//****************************************************************************************************
// Code generated by SFC Generator V1.13 on 13/03/19 17:24:34 by  David Paspa from File G:\Business\Synertec\MPI.SMS\automation\code\awlMaster\stencil\seq_hdr.awl
//****************************************************************************************************
//****************************************************************************************************

//================================ SEQ HEADER ================================//
//            Copyright 2018 Rieckermann Engineering Operations               //
//----------------------------------------------------------------------------//
// Title: UO_MX_SIP                                                       //
//                                                                            //
// Description:                                                               //
// Sequence for Mx sterilise in place operation                                                        //
//                                                                            //
// // SFC Revision History:
// Rev By               Date        CC         Note
// 2.0 David Paspa      27-Nov-2018            Reboot for S7-1500
// 0.3 Srinivas Nimmala 19-May-2010            Wong(Changed Cooling-Preempt)
// 0.2 David Paspa      26-Oct-2009            Added synch flags
// 0.1 Gerald Kontriner 09-Sep-2009            SFC structural design                                                       //
//----------------------------------------------------------------------------//
// Sequencer Revision History:                                                //
// Rev By               Date        CC        Note                            //
// 2.0 David Paspa      05-Jan-2018 NA        Reboot for S7-1500.             //
// 1.6 Khairul Basar    19-Nov-2009 NA        Reset #sqSequencer.STEP.Active  //
//                                            when STEP Finished.             //
// 1.5 Khairul Basar    15-Oct-2009 NA        Placeholder inserted:           //
//                                            "udtSQ_UO";          //
// 1.4 Khairul Basar    06-Oct-2009 NA        R #PAUSE;                       //
// 1.3 Khairul Basar    30-Sep-2009 NA        SEQ_HDR change STEP-0 code      //
//                                            deleted.                        //
// 1.2 Khairul Basar    26-Sep-2009 NA        Refer R4.                       //
// 1.1 Khairul Basar    23-Sep-2009 NA        Refer R3.                       //
// 1.0 Khairul Basar    20-Sep-2009 NA        STEP.Finished flag reset by     //
//                                            JUMP_MAN.                       //
// 0.9 Khairul Basar    11-Sep-2009 NA        SQ_TIMER added as VAR, declared //
//                                            in SEQ_FTR.                     //
// 0.8 Khairul Basar    09-Sep-2009 NA        SqSequencer.Err_Fault is reset  //
//                                            on Stop cmd, Step-0 dead code   //
//                                            deleted from ACT & Verify.      //
//                                            STP_FTR Step_withErr flag       //
//                                            STEP_NUM place holder           //
//                                            configured.                     //
// 0.7 Khairul Basar    28-Aug-2009 NA        SQ_FINISHED OUT added again.    //
//                                            Deleted during major mod R3.    //
// 0.6 Khairul Basar    23-Aug-2009 NA        Refer R2.                       //
// 0.5 Khairul Basar    23-Aug-2009 NA        Refer R1.                       //
// 0.4 Khairul Basar    18-Aug-2009 NA        Reset Step done with/out error  //
//                                            bits using FC:RSET.             //
// 0.3 David Paspa      16-Aug-2009 NA        Added placeholders for header   //
//                                            name and version and revision   //
//                                            history.                        //
// 0.2 Khairul Basar    11-Aug-2009 NA        Retired external udt file for   //
//                                            Static type parameters. All     //
//                                            parameters now IN, OUT or       //
//                                            IN_OUT.                         //
// 0.1 Khairul Basar    12-Jun-2009 NA        Initial design.                 //
//----------------------------------------------------------------------------//
// R4:                                                                        //
// 1.If SQ not finished Resume command will start Step timer, and redo the    //
// last action, verify the feedback.                                          //
// 2."STEP.finished" flag is ANDed with "TRN_AND_JUMP" in the snippet file    //
// TRN_HDR.This is to avoid checking of transition logic if STEP is not       //
// finished yet.                                                              //
// 3.MDCH, Load & transfer typo corrected.                                    //
//                                                                            //
// R3:                                                                        //
// 1.SqStepTimer.IN is reset in STEP_FTR instead of resetting it in TRN_HDR.  //
// This is because TRN_HDTR is not included in the Last step and StepTimer    //
// must reset in the last step.                                               //
// 2.Reset all the timers when SQ stops.Reset done in SEQ_HDR.                //
// Also STEP-finished flag reset when SQ is OFF to                            //
// scan last step.                                                            //
//                                                                            //
// R2:                                                                        //
// 1.Any step error will send the Sequencer into Pause state.Code added in    //
// SEQ_HDR.Snippet Place holder for Bool-array 32 is   //
// deleted.                                                                   //
//                                                                            //
// R1:                                                                        //
// 1.sqStepTimer:All Verification Code must satisfy the condition finish step //
// action within STEP_DELAY time(40s).If step actions not finished within the //
// time period the error flag will raise High signal.Else timer will reset.   //
// 2.sqRunTimer Added therefore can be used as retentive & non retentive.     //
// 3.sqSequencer: This is re-structured UDT which is redefined the symbol     //
// names as well as it gives more clearity.                                   //
// 4.fcMODE and fcCMD functions are added to handle the mode & command        //
// independently regardless of other logic.Two separate UDT udtMODE & udt     //
// CMD assigned to Mode & command function respectively.                      //
// 5.MAN_JUMP programed for manual mode jump operation with or without        //
// Transition code satisfied.TRN_AND_JUMP & NO_VERIFC are the parameters      //
// which will define whether verification code & transition code need to be   //
// checked to perform jump operation.                                         //
// 6.Auto to Manual switchover will be bumpless & will not affect step        //
// operation.Manual to auto switchover can be used to resume Step action at   //
// defined.                                                                   //
// Step number entered in STEPNO_JUMP.                                        //
//                                                                            //
// Parameters:                                                                //
// INPUTS                                                                     //
// ======                                                                     //
// SQ_CMD          Sequence command input inherited from object block         //
//                 0: off/idle                                                //
//                 1: start/initiate                                          //
//                 2: pause                                                   //
//                 3: resume                                                  //
//                 4: reserved (not programmed)                               //
//                 5: reserved (not programmed)                               //
//                 6: abort/go to last step                                   //
//                 7: acknowledge error/fault                                 //
// SQ_MODE         Sequencer Auto/Manual input inherited from object block    //
//                 1: manual                                                  //
//                 2: auto                                                    //
//                                                                            //
// INPUT/OUTPUTS                                                              //
// =============                                                              //
// SQ_JUMP_MAN     Allows manual jumping from one step to the next step. The  //
//                 manual jump flag is ORed with the transition process       //
//                 condition and so can be used to bypass the condition if the//
//                 sequence will not progress.                                //
//                 This input can also be used to jump to any step even       //
//                 when no transition -> step linkage exists. This is only    //
//                 possible when the SQ_MODE is in manual and SQ is in the    //
//                 idle step. The step to jump to is specified in             //
//                 SQ_man_jump_to_step (not accesseble by this FB in/out      //
//                 interface but a separate DB memory location).              //
//                                                                            //
// OUTPUTS                                                                    //
// =======                                                                    //
// SQ_STATE        The calculated state of the sequence                       //
//                 0: off/idle                                                //
//                 1: start/initiated                                         //
//                 2: paused                                                  //
//                 3: resumed                                                 //
//                 4: reserved (wrong Mode)                                   //
//                 5: reserved (Wrong commad)                                 //
//                 6: aborted/go to last step                                 //
//                 7: acknowledged error/fault                                //
// CURSTEP         Current step being proccessed.                             //
// S_ACTIVE        If current step is active                                  //
// NXT_STEP        Next step to jump to if transition condition is true       //
// ERR_FAULT       True if any error/ or fault present                        //
// PAUSED          True if step is paused                                     //
// OFF_IDLE        Sequence is not running but ready for next SQ (in step=0)  //
//----------------------------------------------------------------------------//
// Define variables:                                                          //
//----------------------------------------------------------------------------//
FUNCTION_BLOCK "fbUO_MX_SIP"
TITLE = UO : MX_SIP
{ S7_Optimized_Access := 'TRUE' }
NAME : MUSIP
AUTHOR : REO
VERSION : 2.0

VAR_IN_OUT
    _emv_inlet_state :INT ;	//Vessel inlet sprayballs state
    _vessel_mx :INT ;	//Manufacturing vessel selection M1 or M2
    _emc_gas_pi_vessel_pv :REAL ;	//Vessel pressure
    _emx_drain_state :INT ;	//Device state of emx_drain
    _ema_vessel_state :INT ;	//Device State of ema_vessel
    _emx_mmfl_state :INT ;	//Device state of emx_mmfl
    _emv_vessel_ti_vessel_pv :REAL ;	//TIn105 Vessel Temperature
    _emg_filter_ti_drain_pv :REAL ;	//TIn103 Vent Filter Top Outlet Temperature
    _emt_hex_ti_hex_pv :REAL ;	//TIn109 Heat Exchanger Outlet Temperature
    _emx_drain_ti_drain_pv :REAL ;	//TIn107 Drain Temperature
    _emg_filter_state :INT ;	//Device State of emg_filter
    _emc_water_state :INT ;	//Device State of emc_water
    _emc_gas_state :INT ;	//Device State of emc_gas
    _emv_vessel_state :INT ;	//Device state of emv_vessel

    _emx_mmfl_opened_time :TIME ;	//Time to pulse MMFLx drain valve
    _emc_water_runtime :TIME ;	//Runtime for steam addition. Zero means run forever.
    _emv_inlet_cmd :INT ;	//Vessel inlet sprayballs command
    _emv_inlet_subs :INT ;	//Vessel inlet sprayballs substate
    _emx_drain_cmd :INT ;	//Command to emx_drain
    _emx_drain_subs :INT ;	//Substate selection to emx_drain
    _ema_vessel_cmd :INT ;	//Command to ema_vessel
    _ema_vessel_subs :INT ;	//Substate selection to ema_vessel
    _emx_mmfl_cmd :INT ;	//Command to emx_mmfl
    _emx_mmfl_subs :INT ;	//Substate selection to emx_mmfl
    _emc_water_cmd :INT ;	//Command to emc_water
    _emc_water_subs :INT ;	//Substate selection to emc_water
    _emc_water_medium_liquid :INT ;	//Medium selection to emc_water
    _emc_gas_setpoint :REAL ;	//emc_gas pressure setpoint
    _emg_filter_subs :INT ;	//Substate selection to emg_filter
    _emg_filter_cmd :INT ;	//Command to emg_filter
    _emc_gas_medium_gas :INT ;	//emc_gas_medium
    _emc_gas_subs :INT ;	//Substate selection to emc_gas
    _emv_vessel_subs :INT ;	//Substate selection to emv_vessel
    _emv_vessel_cmd :INT ;	//Command to emv_vessel
    _emc_gas_cmd :INT ;	//Command to emc_gas


    dummy : bool;            // Dummy placeholder for call without comma
END_VAR

VAR
    smc : "udtModeCommandSFC";         // SFC mode and command
    sqStepTimer : "TON";
    sqRunTimer : "fbRunTimer";
    sqSequencer : "udtSFCSequence32";
    SQ_TIMER: "TON";
    SQ_TIMER2: "TON";
    SQ_TIMER3: "TON";
    sqSeqTimerStart : Bool;
    sqSeqTimerStart2 : Bool;
    sqSeqTimerStart3 : Bool;
    sqSeqTimerElapsed : Time;
    sqSeqTimerElapsed2 : Time;
    sqSeqTimerElapsed3 : Time;
    sqSeqTimerExpired : Bool;
    sqSeqTimerExpired2 : Bool;
    sqSeqTimerExpired3 : Bool;
    sqStepTimerElapsed : Time;
    sqStepTimerExpired : Bool;
    _r_time_mmflx_pulse_sip :TIME ;	//Time to pulse MMFLx drain valve during SIP
    _r_time_mmflx_pulse_heat :TIME ;	//Time to pulse MMFLx drain valve during heatup
    _r_pres_gas_empty :REAL ;	//Pressure to empty vessel
    _prompt_try_again :BOOL ;	//UO_MX_SIP Operator to confirm to retry or abort
    _prompt_try_again_confirm_no :BOOL ;	//UO_MX_SIP Operator to confirm to retry or abort confirmed abort
    _prompt_try_again_confirm_yes :BOOL ;	//UO_MX_SIP Operator to confirm to retry or abort confirmed retry
    _log_real_emt_ti_hex_pv :BOOL ;	//UO_MX_SIP HEX Outlet temperature PV
    _log_real_emg_ti_drain_pv :BOOL ;	//UO_MX_SIP Vent filter drain temperature PV
    _log_real_emv_ti_vessel_pv :BOOL ;	//UO_MX_SIP Vessel temperature PV
    _log_real_emx_ti_drain_pv :BOOL ;	//UO_MX_SIP Transfer line drain temperature PV
    _real_emt_ti_hex_pv :REAL ;	//UO_MX_SIP HEX Outlet temperature PV
    _real_emg_ti_drain_pv :REAL ;	//UO_MX_SIP Vent filter drain temperature PV
    _real_emv_ti_vessel_pv :REAL ;	//UO_MX_SIP Vessel temperature PV
    _real_emx_ti_drain_pv :REAL ;	//UO_MX_SIP Transfer line drain temperature PV
    _log_msg_pres_blow_reached :BOOL ;	//UO_MX_SIP Time when HPCA BLOW pressure reached
    _log_msg_pres_leave_reached :BOOL ;	//UO_MX_SIP Time when HPCA LEAVE pressure reached
    _log_msg_sip_timer_reset :BOOL ;	//UO_MX_SIP Sterilisation timer reset
    _log_msg_sip_start :BOOL ;	//UO_MX_SIP Sterilisation begin time
    _log_msg_sip_abort :BOOL ;	//UO_MX_SIP SIP automatic abort due to too many fails
    _log_msg_vacuum_fail_abort :BOOL ;	//UO_MX_SIP Operator confirmed to abort when sterilisation vacuum failed
    _log_msg_vacuum_fail_repeat :BOOL ;	//UO_MX_SIP Operator confirmed to retry when sterilisation vacuum failed
    _log_msg_vacuum_fail :BOOL ;	//UO_MX_SIP Sterilisation vacuum failed
    _log_msg_steam_closed :BOOL ;	//UO_MX_SIP Steam closed time
    _log_real_positive_pressure :BOOL ;	//UO_MX_SIP Positive pressure reached
    _log_msg_steam_open :BOOL ;	//UO_MX_SIP Steam opened time
    _log_msg_vacuum_begin :BOOL ;	//UO_MX_SIP Vacuum begin time
    _log_msg_sip_begin :BOOL ;	//UO_MX_SIP begin time
    _log_msg_sip_end :BOOL ;	//UO_MX_SIP end time
    _log_msg_sip_complete :BOOL ;	//UO_MX_SIP Sterilisation end time
    _r_pulse_number :INT ;	//MX SIP Number of times to pulse SIP drain valves
    _pulse_counter :INT ;	//counter pulse_vlv
    _r_num_sip_abort :INT ;	//MX SIP Number of SIP attempts before abort
    _ctr_sip_abort :INT ;	//counter of SIP abort times
    _r_time_sip :TIME ;	//MX SIP Sterilisation time
    _sip_timer_started :BOOL ;	//sip_timer_started
    _r_time_sip_abort :TIME ;	//MX SIP Time to abort SIP if sterilisation temperature not reached
    _r_time_stm_drain_mx :TIME ;	//MX SIP Time to steam drain valves
    _r_time_eject :TIME ;	//MX SIP Vacuum system run time before timeout
    _r_pres_vac :REAL ;	//MX SIP Vacuum pressure setpoint
    _r_temp_sip :REAL ;	//MX SIP Sterilisation temperature
    _r_temp_sip_vent :REAL ;	//MX SIP Sterilisation temperature for vessel vent valve line
    _log_disconnect :BOOL ;	//UO_MX_SIP Operator confirmed all vessel pipe entries are disconnected.
    _real_positive_pressure :REAL ;	//UO_MX_SIP Positive pressure reached
    _r_time_drain_pulse :TIME ;	//MX SIP Time to pulse drain valves
    _r_pres_hpca_leave :REAL ;	//MX SIP HPCA pressure after condensate drain blow down
    _r_pres_hpca_blow :REAL ;	//MX SIP HPCA Pressure to blow out condesate drain valves
    _r_pres_lpca_blanket :REAL ;	//MX SIP LPCA blanket pressure
    _r_pres_stm_pos :REAL ;	//MX SIP Positive steam pressure threshold

END_VAR

BEGIN
NETWORK
TITLE =Call Mode checking function
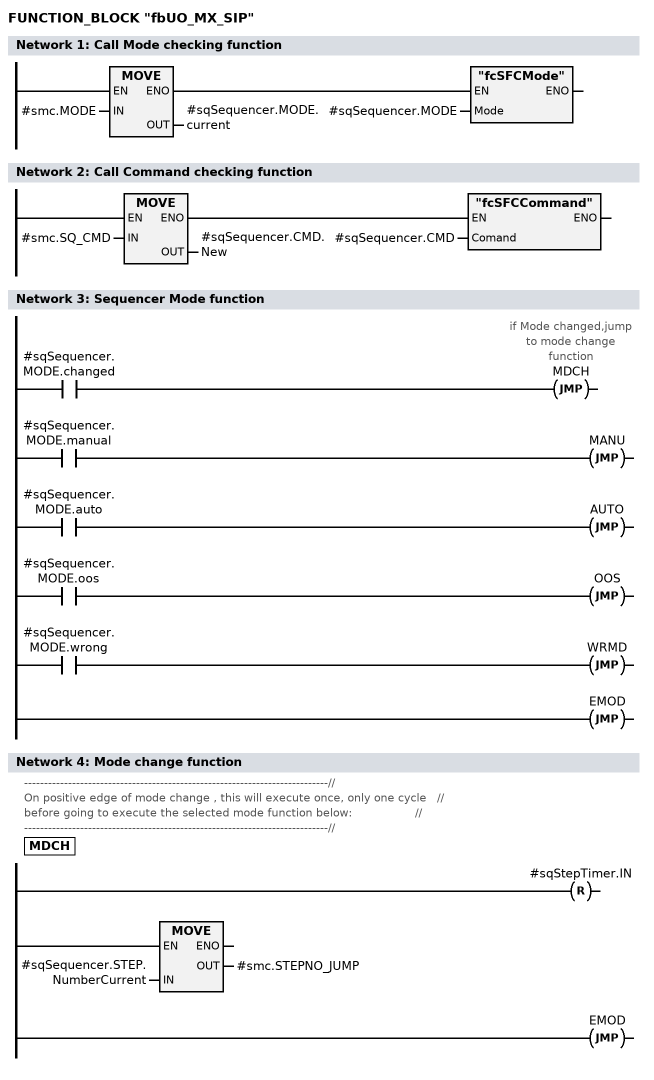
    L     #smc.MODE;
    T     #sqSequencer.MODE.current;
    CALL "fcSFCMode"
    (   Mode                 := #sqSequencer.MODE
    );

NETWORK
TITLE =Call Command checking function
    L     #smc.SQ_CMD;
    T     #sqSequencer.CMD.New;
    CALL "fcSFCCommand"
    (   Comand               := #sqSequencer.CMD
    );

NETWORK
TITLE =Sequencer Mode function

      A     #sqSequencer.MODE.changed;
      JC    MDCH; // if Mode changed,jump to mode change function
      A     #sqSequencer.MODE.manual;
      JC    MANU;
      A     #sqSequencer.MODE.auto;
      JC    AUTO;
      A     #sqSequencer.MODE.oos;
      JC    OOS;
      A     #sqSequencer.MODE.wrong;
      JC    WRMD;
      JU    EMOD;

NETWORK
TITLE =Mode change function
//----------------------------------------------------------------------------//
// On positive edge of mode change , this will execute once, only one cycle   //
// before going to execute the selected mode function below:                  //
//----------------------------------------------------------------------------//
MDCH: NOP   0;
      SET   ;
      R     #sqStepTimer.IN;
      L     #sqSequencer.STEP.NumberCurrent;
      T     #smc.STEPNO_JUMP;
      JU    EMOD;

NETWORK
TITLE =Manual Mode function
//----------------------------------------------------------------------------//
// #TRN_AND_JUMP=can set/reset                                                //
// #sqSequencer.STEP.JumpCtrl=Can set/reset by #MAN_JUMP                      //
// #NO_VERIFIC=Can set/ Reset                                                 //
//----------------------------------------------------------------------------//
MANU: NOP   0; //Manual mode selected



      A     #smc.MAN_JUMP;
      =     #sqSequencer.STEP.JumpCtrl;
      A     #smc.MAN_JUMP;
      JCN   EMOD;

      L     #smc.STEPNO_JUMP;
      T     #sqSequencer.STEP.NumberNext;
      T     #sqSequencer.STEP.NumberCurrent;
      R     #smc.MAN_JUMP; //Reset MAN_JUMP after loading user destination Step number
      R     #sqSequencer.STEP.Finished; //Reset finish flag, to execute next step action
      JU    EMOD;

NETWORK
TITLE =Auto Mode function
//----------------------------------------------------------------------------//
// #TRN_AND_JUMP=always set                                                   //
// #sqSequencer.STEP.JumpCtrl=Always set                                      //
// #NO_VERIFIC=Alwasy Reset                                                   //
//----------------------------------------------------------------------------//
AUTO: NOP   0; //Auto mode selected



      R     #smc.MAN_JUMP;
      S     #smc.TRN_AND_JUMP;
      R     #smc.NO_VERIFIC;
      S     #sqSequencer.STEP.JumpCtrl; //Always Set in auto mode

      L     #sqSequencer.STEP.NumberCurrent;
      T     #smc.STEPNO_JUMP;
      JU    EMOD;
NETWORK
TITLE =OOS mode function

OOS:  NOP   0; // Out of service
      JU    EMOD;
WRMD: NOP   0; //Wrong mode selected
      S     #sqSequencer.Error_Fault;
      L     "dbCONST".SEQ.STATE.WRMODE;
      T     #smc.SQ_STATE;

      JU    EMOD;

NETWORK
TITLE =Mode not changedd

      NOP   0;

NETWORK
TITLE =End Mode function

EMOD: NOP   0;

NETWORK
TITLE =An error will Pause the Sequencer,Operator must Resume SQ to run

      A     #sqSequencer.Error_Fault;
      AN    #sqSequencer.CMD.Changed;
      JC    PAUS;

NETWORK
TITLE =Command Action function

      A     #sqSequencer.CMD.Changed;
      JCN   CNCH; // if Command not changed,jump to end function
      R     #sqStepTimer.IN;

      A     #sqSequencer.CMD.Start;
      JC    STRT;

      A     #sqSequencer.CMD.Stop;
      JC    STOP;

      A     #sqSequencer.CMD.Pause;
      JC    PAUS;

      A     #sqSequencer.CMD.Resume;
      JC    RESM;

      A     #sqSequencer.CMD.Abort;
      JC    _abrt_begin;

      A     #sqSequencer.CMD.Ack;
      JC    ACKN;

      A     #sqSequencer.CMD.wrong;
      JC    WCMD;

      JU    ECMD; //Wrong command/not specified command
//End Comand function

NETWORK
TITLE =Comand -Start/Initiate action function

STRT: NOP   0;
      R     #smc.OFF_IDLE;
      R     #smc.ABORTED;
      R     #smc.PAUSED;
      R     #sqSequencer.STEP.Active;
      R     #sqSequencer.STEP.Finished;
      R     #sqSequencer.STEP.ActionFinished;
      R     #sqSequencer.STEP.Jump;
      R     #sqSequencer.STEP.TimerExpired;
      R     #sqSequencer.STEP.Error_Fault;
      R     #sqSequencer.STEP.ActionVerified;
      R     #sqStepTimer.IN;

//      S     #sqRunTimer.RESET;

//----------------------------------------------------------------------------//
// Load Initial step Number:                                                  //
//----------------------------------------------------------------------------//
      L     1;
      T     #sqSequencer.STEP.Initial;
      L     #sqSequencer.STEP.Initial;
      T     #sqSequencer.STEP.NumberCurrent;
      T     #sqSequencer.STEP.NumberNext;

      L     "dbCONST".SEQ.STATE.STARTED;
      T     #smc.SQ_STATE;

NETWORK
TITLE = Reset sequence Done bits
    //------------------------------------------------------------------------//
    // Reset Step done bits:                                                  //
    //------------------------------------------------------------------------//
    CALL FILL_BLK
    {value_type := 'Bool', count_type := 'UInt'}
    (   IN                   := 0 ,
        COUNT                := 32 ,
        OUT                  := #sqSequencer.STEP.Done[1]
    );

NETWORK
TITLE = Reset sequence Error bits
    //------------------------------------------------------------------------//
    // Reset Step error bits:                                                 //
    //------------------------------------------------------------------------//
    CALL FILL_BLK
    {value_type := 'Bool', count_type := 'UInt'}
    (   IN                   := 0 ,
        COUNT                := 32 ,
        OUT                  := #sqSequencer.STEP.WithError[1]
    );

    JU    ECMD; //End Function

NETWORK
TITLE =Comand -Stop action function

STOP: NOP   0;
      S     #smc.OFF_IDLE;
      R     #sqSequencer.STEP.Active;
      R     #sqSequencer.STEP.Finished;
      R     #sqSequencer.STEP.ActionFinished;
      R     #sqSequencer.STEP.Jump;
      R     #sqSequencer.STEP.TimerExpired;
      R     #sqSequencer.STEP.Error_Fault;
      R     #sqSequencer.Error_Fault;
      R     #sqSequencer.STEP.ActionVerified;
      R     #sqRunTimer.ENABLE;
      R     #sqStepTimer.IN;
      R     #sqSeqTimerStart;
      R     #sqSeqTimerStart2;
      R     #sqSeqTimerStart3;
      R     #smc.PAUSED;
      R     #smc.ABORTED;


//Go to last step
      L     25;
      T     #sqSequencer.FinalStep;
      T     #sqSequencer.STEP.NumberNext;

      JU    ECMD; //End Function

NETWORK
TITLE =Comand -Pause action function

PAUS: NOP   0;
      S     #smc.PAUSED;
      R     #smc.S_ACTIVE;
      S     #sqRunTimer.PAUSE;
      L     #sqSequencer.STEP.NumberCurrent;
      T     #smc.STEPNO_JUMP;
      L     "dbCONST".SEQ.STATE.PAUSED;
      T     #smc.SQ_STATE;

      JU    ECMD; //End Function

NETWORK
TITLE =Comand -Resume action function

RESM: NOP   0;
      R     #smc.PAUSED;
      R     #sqRunTimer.PAUSE;
      R     #sqStepTimer.IN; //Reset Step timer
      L     "dbCONST".SEQ.STATE.RESUMED;
      T     #smc.SQ_STATE;

      A     #smc.SQ_FINISHED;
      JC    ECMD;
      R     #sqSequencer.STEP.Active;
      R     #sqSequencer.STEP.Finished;
      R     #sqSequencer.STEP.ActionFinished;

      JU    ECMD; //End Function

NETWORK
TITLE =Comand -Abort action function

_abrt_begin: NOP   0;

      S     #smc.ABORTED;
      R     #sqSequencer.STEP.Active;
      R     #sqSequencer.STEP.Finished;
      R     #sqSequencer.STEP.ActionFinished;
      R     #sqSequencer.STEP.Jump;
      R     #sqSequencer.STEP.TimerExpired;
      R     #sqSequencer.STEP.Error_Fault;
      R     #sqSequencer.Error_Fault;
      R     #sqSequencer.STEP.ActionVerified;
      R     #sqRunTimer.ENABLE;
      R     #sqStepTimer.IN;
      R     #sqSeqTimerStart;
      R     #sqSeqTimerStart2;
      R     #sqSeqTimerStart3;
      R     #smc.PAUSED;
      R     #smc.OFF_IDLE;


//Go to last step
      L     25;
      T     #sqSequencer.FinalStep;
      T     #sqSequencer.STEP.NumberNext;

      JU    ECMD;

NETWORK
TITLE =Comand -Acknowledge action function

ACKN: NOP   0;
      R     #smc.ERR_FAULT;
      R     #sqSequencer.Error_Fault;
      L     "dbCONST".SEQ.STATE.ACKNOWLEDGED;
      T     #smc.SQ_STATE;

      JU    ECMD; //End Function

NETWORK
TITLE =Comand -wrong/unavailable

WCMD: NOP   0;

      S     #sqSequencer.Error_Fault;
      L     "dbCONST".SEQ.STATE.WRCMD;
      T     #smc.SQ_STATE;

      JU    ECMD;
NETWORK
TITLE =Comand -not changedd

CNCH: NOP   0; // Command not changed

NETWORK
TITLE =End command Function

ECMD: NOP   0;

NETWORK
TITLE =Sequencer Step Jump distrubution list
    //------------------------------------------------------------------------//
    // Sequencer step jump list. Load the step number to execute the step:    //
    //------------------------------------------------------------------------//
    L     #sqSequencer.STEP.NumberCurrent;
    JL    SQER; // If Sequencer Step number invalid or greater than available number of step
    JU    S000; // Exceptional Error Handling
    JU    S001; // STEP-001:
JU    S002; // STEP-002:
JU    S003; // STEP-003:
JU    S004; // STEP-004:
JU    S005; // STEP-005:
JU    S006; // STEP-006:
JU    S007; // STEP-007:
JU    S008; // STEP-008:
JU    S009; // STEP-009:
JU    S010; // STEP-010:
JU    S011; // STEP-011:
JU    S012; // STEP-012:
JU    S013; // STEP-013:
JU    S014; // STEP-014:
JU    S015; // STEP-015:
JU    S016; // STEP-016:
JU    S017; // STEP-017:
JU    S018; // STEP-018:
JU    S019; // STEP-019:
JU    S020; // STEP-020:
JU    S021; // STEP-021:
JU    S022; // STEP-022:
JU    S023; // STEP-023:
JU    S024; // STEP-024:
JU    S025; // STEP-025:


    //------------------------------------------------------------------------//
    // If Step number is Invalid or Out of Range:                             //
    //------------------------------------------------------------------------//
SQER: NOP   0;
    A     "alwaysLow";
    S     #sqSequencer.Error_Fault;
    JU    COMM; // Jump to Common Sequencer code handling function

NETWORK
TITLE =STEP0 STEP0 STEP0 STEP0 STEP0 STEP0 STEP0 STEP0 STEP0 STEP0 STEP
    //------------------------------------------------------------------------//
    // STEP0 STEP0 STEP0 STEP0 STEP0 STEP0 STEP0 STEP0 STEP0 STEP0 STEP0 STEP //
    // AUTOCODE   AUTOCODE   AUTOCODE   AUTOCODE   AUTOCODE   AUTOCODE   AUTO //
    // STEP0 STEP0 STEP0 STEP0 STEP0 STEP0 STEP0 STEP0 STEP0 STEP0 STEP0 STEP //
    //------------------------------------------------------------------------//

NETWORK
TITLE =S000: STEP0::If Paused exit

S000: NOP   0;
      JU    COMM;






NETWORK
TITLE =S001: STEP-01::UO_MX_SIP : Unit operation started
    //================================ STEP HEADER ===========================//
    // STEP001 STEP001 STEP001 STEP001
    // AUTOCODE   AUTOCODE   AUTOCODE   AUTOCODE   AUTOCODE   AUTOCODE   AUTO //
    // STEP001 STEP001 STEP001 STEP001
    //------------------------------------------------------------------------//
    // Open Mx outlet and MMFL transfer line valves to drain vessel.
    //------------------------------------------------------------------------//
S001: NOP   0;

      SET;
      R     #sqSequencer.STEP.jumpDone[01];
      A     #sqSequencer.CMD.Pause; //If paused jump
      JC    COMM;

NETWORK
TITLE =S001:STEP-01:Begin Action

      A     #sqSequencer.STEP.Finished;
      JC    A001; // Exit Action code, Jump to A001 Transition code

      //----------------------------------------------------------------------//
      // Begin step Action:                                                   //
      //----------------------------------------------------------------------//
      A     #sqSequencer.STEP.Active;
      JC    L001; // Action number loaded, Jump to L001--Step Action List

      //----------------------------------------------------------------------//
      // Load Default/Initial Step action number:                             //
      //----------------------------------------------------------------------//
      S     #sqSequencer.STEP.Active;
      S     #sqStepTimer.IN;
      L     1; //First Action, Step must contain Minimum one action
      T     #sqSequencer.STEP.ActionNumber;

//----------------------------------------------------------------------------//
// Step action list.                                                          //
// aann=mini Action step number(aa) inside main step number(nn)               //
// First Action aa00, Second action ab00, Third ac00, etc.                    //
//----------------------------------------------------------------------------//
L001: NOP   0;

      L     #sqSequencer.STEP.ActionNumber;
      JL    r001; //Wrong Action number
      JU    _001; //Action error handling
       JU    aa01; //ACTION-01
JU    ab01; //ACTION-02


//----------------------------------------------------------------------------//
// More step action in the list can be inserted here, upto ab is tested:      //
//----------------------------------------------------------------------------//
r001: NOP   0; //Wrong action number
      S     #sqSequencer.Error_Fault;
      JU    k001; //Exit
_001: NOP   0; // Action error handling
      JU    k001; // Exit






NETWORK
TITLE =S001:: STEP-001:: : ACTION CODE
    //================================ ACT HEADER ============================//
    // ACTION ACTION ACTION ACTION ACTION ACTION ACTION ACTION ACTION ACTION  //
    // AUTOCODE   AUTOCODE   AUTOCODE   AUTOCODE   AUTOCODE   AUTOCODE   AUTO //
    // ACTION ACTION ACTION ACTION ACTION ACTION ACTION ACTION ACTION ACTION  //
    //------------------------------------------------------------------------//
    // //Reset EMs
    aa01: NOP   0;

    //------------------------------------------------------------------------//
    // ACT ACT ACT ACT ACT ACT ACT ACT ACT ACT ACT ACT ACT ACT ACT ACT ACT    //
    //------------------------------------------------------------------------//
    //Log SIP operation begin time.
SET;
S #_log_msg_sip_begin;


L "dbCONST".BLK.CMD.STOP;
T #_emv_inlet_cmd;
T #_emv_vessel_cmd;
T #_emx_mmfl_cmd;

    //------------------------------------------------------------------------//
    // VERIFY  VERIFY VERIFY VERIFY VERIFY VERIFY VERIFY VERIFY VERIFY VERIFY //
    //------------------------------------------------------------------------//
    //Verify emv_inlet stopped.
A(;
L    #_emv_inlet_state;
L    "dbCONST".BLK.STATE.STOPPED;
==I;
);
//Verify emv_vessel stopped.
A(;
L    #_emv_vessel_state;
L    "dbCONST".BLK.STATE.STOPPED;
==I;
);
//Verify if emx_mmfl stopped.
A(;
L   #_emx_mmfl_state;
L    "dbCONST".BLK.STATE.STOPPED;
==I;
);

    S     #sqSequencer.STEP.ActionVerified; //Action verified

    //------------------------------------------------------------------------//
    // Action done:                                                           //
    //------------------------------------------------------------------------//
    O     #sqSequencer.STEP.ActionVerified;
    O     #smc.NO_VERIFIC;       //No verification , bypass verification code
    S     #sqSequencer.STEP.ActionFinished;






    //============================= ACT FOOTER ===============================//
    // AUTOCODE   AUTOCODE   AUTOCODE   AUTOCODE   AUTOCODE   AUTOCODE   AUTO //
    // Get Ready after action finished:                                       //
    //------------------------------------------------------------------------//
    A     #sqSequencer.STEP.ActionFinished;
    JCN   k001;

    //------------------------------------------------------------------------//
    // Reset Action finished flag, ready for next step action:                //
    //------------------------------------------------------------------------//
    R     #sqSequencer.STEP.ActionVerified;
    R     #sqSequencer.STEP.ActionFinished;

    //------------------------------------------------------------------------//
    // Load Next Step Action number:                                          //
    //------------------------------------------------------------------------//
    L     02; //Load next Action
    T     #sqSequencer.STEP.ActionNumber;






NETWORK
TITLE =S001:: STEP-001:: : ACTION CODE
    //================================ ACT HEADER ============================//
    // ACTION ACTION ACTION ACTION ACTION ACTION ACTION ACTION ACTION ACTION  //
    // AUTOCODE   AUTOCODE   AUTOCODE   AUTOCODE   AUTOCODE   AUTOCODE   AUTO //
    // ACTION ACTION ACTION ACTION ACTION ACTION ACTION ACTION ACTION ACTION  //
    //------------------------------------------------------------------------//
    // //Open valves for steaming
    ab01: NOP   0;

    //------------------------------------------------------------------------//
    // ACT ACT ACT ACT ACT ACT ACT ACT ACT ACT ACT ACT ACT ACT ACT ACT ACT    //
    //------------------------------------------------------------------------//
    //Open Mx inlet valves.
L "dbCONST".BLK.EMV2.SUBS.CHARGE;
T #_emv_inlet_subs;
L "dbCONST".BLK.CMD.START;
T #_emv_inlet_cmd;

//Open Mx outlet valve.
L "dbCONST".BLK.EMV1.SUBS.DISCHARGE;
T #_emv_vessel_subs;
L "dbCONST".BLK.CMD.START;
T #_emv_vessel_cmd;

// Set emx_mmfl to substate SIP and start it.
L "dbCONST".BLK.EMX1.SUBS.SIP;
T #_emx_mmfl_subs;
L "dbCONST".BLK.CMD.START;
T #_emx_mmfl_cmd;


    //------------------------------------------------------------------------//
    // VERIFY  VERIFY VERIFY VERIFY VERIFY VERIFY VERIFY VERIFY VERIFY VERIFY //
    //------------------------------------------------------------------------//
    //Verify emv_inlet changed to substate CHARGE.
A(;
L    #_emv_inlet_subs;
L    "dbCONST".BLK.EMV2.SUBS.CHARGE;
==I;
);
//Verify emv_vessel changed to substate DISCHARGE.
A(;
L    #_emv_vessel_subs;
L    "dbCONST".BLK.EMV1.SUBS.DISCHARGE;
==I;
);
//Verify if emx_mmfl changed to substate SIP.
A(;
L   #_emx_mmfl_subs;
L   "dbCONST".BLK.EMX1.SUBS.SIP;
==I;
);
    S     #sqSequencer.STEP.ActionVerified; //Action verified

    //------------------------------------------------------------------------//
    // Action done:                                                           //
    //------------------------------------------------------------------------//
    O     #sqSequencer.STEP.ActionVerified;
    O     #smc.NO_VERIFIC;       //No verification , bypass verification code
    S     #sqSequencer.STEP.ActionFinished;






    //============================= STEP FOOTER ==============================//
    // AUTOCODE   AUTOCODE   AUTOCODE   AUTOCODE   AUTOCODE   AUTOCODE   AUTO //
    // Get Ready after action finished:                                       //
    //------------------------------------------------------------------------//
    A     #sqSequencer.STEP.ActionFinished;
    JCN   k001;

    //------------------------------------------------------------------------//
    // Reset Action finished flag, ready for next step action:                //
    //------------------------------------------------------------------------//
    R     #sqSequencer.STEP.ActionVerified;
    R     #sqSequencer.STEP.ActionFinished;

    //------------------------------------------------------------------------//
    // If ALL actions are finished:                                           //
    //------------------------------------------------------------------------//
    SET   ;
    S     #sqSequencer.STEP.Finished;
    R     #sqSequencer.STEP.Active;
    S     #sqSequencer.STEP.Done[01];

    //------------------------------------------------------------------------//
    // End Step action(s):                                                    //
    //------------------------------------------------------------------------//
    JU    k001;

//----------------------------------------------------------------------------//
// Finished Step Action(s):                                                   //
//----------------------------------------------------------------------------//
k001: NOP   0;

    A     #sqStepTimerExpired;
    S     #sqSequencer.STEP.WithError[01]; // Step error flag
    S     #sqSequencer.Error_Fault;
    R     #sqStepTimer.IN;

NETWORK
TITLE =S001:STEP-001::Begin Transition
    //------------------------------------------------------------------------//
    // Begin the transition code:                                             //
    //------------------------------------------------------------------------//
    A001: NOP   0;
    R     #sqStepTimer.IN;






    //============================= TRAN HEADER ==============================//
    // AUTOCODE   AUTOCODE   AUTOCODE   AUTOCODE   AUTOCODE   AUTOCODE   AUTO //
    // Bypass transition if manual jump:                                      //
    //------------------------------------------------------------------------//
    A     #sqSequencer.STEP.Finished;
    A     #smc.TRN_AND_JUMP;     //Manual jump is set Transition as bypassed
    JCN   COMM;              //exit

NETWORK
TITLE =S001::STEP 001:TRAN 001: Empty Transition
//----------------------------------------------------------------------------//
// TRAN   TRAN   TRAN   TRAN   TRAN   TRAN   TRAN   TRAN   TRAN   TRAN   TRAN //
// TRAN   TRAN   TRAN   TRAN   TRAN   TRAN   TRAN   TRAN   TRAN   TRAN   TRAN //
//----------------------------------------------------------------------------//
// Empty Transition
//----------------------------------------------------------------------------//
// CONDITION   CONDITION   CONDITION   CONDITION   CONDITION   CONDITION   CO //
// CONDITION   CONDITION   CONDITION   CONDITION   CONDITION   CONDITION   CO //
//----------------------------------------------------------------------------//
A "uncondJump";






    //============================= TRAN FOOTER ==============================//
    // Transition jump control:                                               //
    //------------------------------------------------------------------------//
    A     #sqSequencer.STEP.JumpCtrl;
    S     #sqSequencer.STEP.Jump;
    S     #sqSequencer.STEP.jumpDone[01];

NETWORK
TITLE =S001:t001::TRANS-v: EXIT TRANSITION AND READY THE NEXT STEP
    //------------------------------------------------------------------------//
    // Check the jump flag and jump to the next step if the transition        //
    // condition is true and has set the jump flag:                           //
    //------------------------------------------------------------------------//
    A     #sqSequencer.STEP.Jump;
    JCN   x001;

    R     #sqSequencer.STEP.Jump;
    R     #sqSequencer.STEP.Finished;

    L     02;     // Load next STEPNO to jump to if transition satisfied
    T     #sqSequencer.STEP.NumberNext; //Next Step02.

    JU    COMM;              // Transition satisfied, Exit, go to next step
x001: NOP   0;






NETWORK
TITLE =S001::STEP-001:EXIT TRANSITION:
    //========================== STEP TRANSFER ===============================//
    // Jump to the common step progression code:                              //
    //------------------------------------------------------------------------//
    JU    COMM;






NETWORK
TITLE =S002: STEP-02::UO_MX_SIP : Vacuum Operation Commenced
    //================================ STEP HEADER ===========================//
    // STEP002 STEP002 STEP002 STEP002
    // AUTOCODE   AUTOCODE   AUTOCODE   AUTOCODE   AUTOCODE   AUTOCODE   AUTO //
    // STEP002 STEP002 STEP002 STEP002
    //------------------------------------------------------------------------//
    // Set other Mx equipments to SAFE state.
    //
    // Enable vacuum and start vacuum timer(time_eject). Log vacuum start time
    //------------------------------------------------------------------------//
S002: NOP   0;

      SET;
      R     #sqSequencer.STEP.jumpDone[02];
      A     #sqSequencer.CMD.Pause; //If paused jump
      JC    COMM;

NETWORK
TITLE =S002:STEP-02:Begin Action

      A     #sqSequencer.STEP.Finished;
      JC    A002; // Exit Action code, Jump to A002 Transition code

      //----------------------------------------------------------------------//
      // Begin step Action:                                                   //
      //----------------------------------------------------------------------//
      A     #sqSequencer.STEP.Active;
      JC    L002; // Action number loaded, Jump to L002--Step Action List

      //----------------------------------------------------------------------//
      // Load Default/Initial Step action number:                             //
      //----------------------------------------------------------------------//
      S     #sqSequencer.STEP.Active;
      S     #sqStepTimer.IN;
      L     1; //First Action, Step must contain Minimum one action
      T     #sqSequencer.STEP.ActionNumber;

//----------------------------------------------------------------------------//
// Step action list.                                                          //
// aann=mini Action step number(aa) inside main step number(nn)               //
// First Action aa00, Second action ab00, Third ac00, etc.                    //
//----------------------------------------------------------------------------//
L002: NOP   0;

      L     #sqSequencer.STEP.ActionNumber;
      JL    r002; //Wrong Action number
      JU    _002; //Action error handling
       JU    aa02; //ACTION-01
JU    ab02; //ACTION-02


//----------------------------------------------------------------------------//
// More step action in the list can be inserted here, upto ab is tested:      //
//----------------------------------------------------------------------------//
r002: NOP   0; //Wrong action number
      S     #sqSequencer.Error_Fault;
      JU    k002; //Exit
_002: NOP   0; // Action error handling
      JU    k002; // Exit






NETWORK
TITLE =S002:: STEP-002:: : ACTION CODE
    //================================ ACT HEADER ============================//
    // ACTION ACTION ACTION ACTION ACTION ACTION ACTION ACTION ACTION ACTION  //
    // AUTOCODE   AUTOCODE   AUTOCODE   AUTOCODE   AUTOCODE   AUTOCODE   AUTO //
    // ACTION ACTION ACTION ACTION ACTION ACTION ACTION ACTION ACTION ACTION  //
    //------------------------------------------------------------------------//
    // //Set other Mx equipment to SAFE state.
    aa02: NOP   0;

    //------------------------------------------------------------------------//
    // ACT ACT ACT ACT ACT ACT ACT ACT ACT ACT ACT ACT ACT ACT ACT ACT ACT    //
    //------------------------------------------------------------------------//
    L "dbCONST".BLK.CMD.STOP;
T  #_ema_vessel_cmd;
T  #_emc_gas_cmd;
T  #_emc_water_cmd;

    //------------------------------------------------------------------------//
    // VERIFY  VERIFY VERIFY VERIFY VERIFY VERIFY VERIFY VERIFY VERIFY VERIFY //
    //------------------------------------------------------------------------//
    A(;
L #_ema_vessel_state;
L "dbCONST".BLK.STATE.STOPPED;
==I;
);
A(;
L #_emc_gas_state;
L "dbCONST".BLK.STATE.STOPPED;
==I;
);
A(;
L #_emc_water_state;
L "dbCONST".BLK.STATE.STOPPED;
==I;
);
    S     #sqSequencer.STEP.ActionVerified; //Action verified

    //------------------------------------------------------------------------//
    // Action done:                                                           //
    //------------------------------------------------------------------------//
    O     #sqSequencer.STEP.ActionVerified;
    O     #smc.NO_VERIFIC;       //No verification , bypass verification code
    S     #sqSequencer.STEP.ActionFinished;






    //============================= ACT FOOTER ===============================//
    // AUTOCODE   AUTOCODE   AUTOCODE   AUTOCODE   AUTOCODE   AUTOCODE   AUTO //
    // Get Ready after action finished:                                       //
    //------------------------------------------------------------------------//
    A     #sqSequencer.STEP.ActionFinished;
    JCN   k002;

    //------------------------------------------------------------------------//
    // Reset Action finished flag, ready for next step action:                //
    //------------------------------------------------------------------------//
    R     #sqSequencer.STEP.ActionVerified;
    R     #sqSequencer.STEP.ActionFinished;

    //------------------------------------------------------------------------//
    // Load Next Step Action number:                                          //
    //------------------------------------------------------------------------//
    L     02; //Load next Action
    T     #sqSequencer.STEP.ActionNumber;






NETWORK
TITLE =S002:: STEP-002:: : ACTION CODE
    //================================ ACT HEADER ============================//
    // ACTION ACTION ACTION ACTION ACTION ACTION ACTION ACTION ACTION ACTION  //
    // AUTOCODE   AUTOCODE   AUTOCODE   AUTOCODE   AUTOCODE   AUTOCODE   AUTO //
    // ACTION ACTION ACTION ACTION ACTION ACTION ACTION ACTION ACTION ACTION  //
    //------------------------------------------------------------------------//
    // //Enable vacuum and start vacuum timer. Log Vacuum begin time
    ab02: NOP   0;

    //------------------------------------------------------------------------//
    // ACT ACT ACT ACT ACT ACT ACT ACT ACT ACT ACT ACT ACT ACT ACT ACT ACT    //
    //------------------------------------------------------------------------//
    //Enable vacuum.
L "dbCONST".SEL.GAS.VACUUM;
T #_emc_gas_medium_gas;
L "dbCONST".BLK.EMC1.SUBS.VALVE;
T #_emc_gas_subs;
L "dbCONST".BLK.CMD.START;
T #_emc_gas_cmd;

// Start vacuum timer
A #SQ_TIMER.Q;
R #sqSeqTimerStart;

AN #SQ_TIMER.Q;
S #sqSeqTimerStart;
L #_r_time_eject;
L 1000;
*I;
T #SQ_TIMER.PT;

//Log vacuum begin time.
SET;
S #_log_msg_vacuum_begin;

    //------------------------------------------------------------------------//
    // VERIFY  VERIFY VERIFY VERIFY VERIFY VERIFY VERIFY VERIFY VERIFY VERIFY //
    //------------------------------------------------------------------------//
    A #sqSeqTimerStart;
    S     #sqSequencer.STEP.ActionVerified; //Action verified

    //------------------------------------------------------------------------//
    // Action done:                                                           //
    //------------------------------------------------------------------------//
    O     #sqSequencer.STEP.ActionVerified;
    O     #smc.NO_VERIFIC;       //No verification , bypass verification code
    S     #sqSequencer.STEP.ActionFinished;






    //============================= STEP FOOTER ==============================//
    // AUTOCODE   AUTOCODE   AUTOCODE   AUTOCODE   AUTOCODE   AUTOCODE   AUTO //
    // Get Ready after action finished:                                       //
    //------------------------------------------------------------------------//
    A     #sqSequencer.STEP.ActionFinished;
    JCN   k002;

    //------------------------------------------------------------------------//
    // Reset Action finished flag, ready for next step action:                //
    //------------------------------------------------------------------------//
    R     #sqSequencer.STEP.ActionVerified;
    R     #sqSequencer.STEP.ActionFinished;

    //------------------------------------------------------------------------//
    // If ALL actions are finished:                                           //
    //------------------------------------------------------------------------//
    SET   ;
    S     #sqSequencer.STEP.Finished;
    R     #sqSequencer.STEP.Active;
    S     #sqSequencer.STEP.Done[02];

    //------------------------------------------------------------------------//
    // End Step action(s):                                                    //
    //------------------------------------------------------------------------//
    JU    k002;

//----------------------------------------------------------------------------//
// Finished Step Action(s):                                                   //
//----------------------------------------------------------------------------//
k002: NOP   0;

    A     #sqStepTimerExpired;
    S     #sqSequencer.STEP.WithError[02]; // Step error flag
    S     #sqSequencer.Error_Fault;
    R     #sqStepTimer.IN;

NETWORK
TITLE =S002:STEP-002::Begin Transition
    //------------------------------------------------------------------------//
    // Begin the transition code:                                             //
    //------------------------------------------------------------------------//
    A002: NOP   0;
    R     #sqStepTimer.IN;






    //============================= TRAN HEADER ==============================//
    // AUTOCODE   AUTOCODE   AUTOCODE   AUTOCODE   AUTOCODE   AUTOCODE   AUTO //
    // Bypass transition if manual jump:                                      //
    //------------------------------------------------------------------------//
    A     #sqSequencer.STEP.Finished;
    A     #smc.TRN_AND_JUMP;     //Manual jump is set Transition as bypassed
    JCN   COMM;              //exit

NETWORK
TITLE =S002::STEP 002:TRAN 002: Pressure below setpoint?
//----------------------------------------------------------------------------//
// TRAN   TRAN   TRAN   TRAN   TRAN   TRAN   TRAN   TRAN   TRAN   TRAN   TRAN //
// TRAN   TRAN   TRAN   TRAN   TRAN   TRAN   TRAN   TRAN   TRAN   TRAN   TRAN //
//----------------------------------------------------------------------------//
// Pressure reduced below PRES_VAC.
//----------------------------------------------------------------------------//
// CONDITION   CONDITION   CONDITION   CONDITION   CONDITION   CONDITION   CO //
// CONDITION   CONDITION   CONDITION   CONDITION   CONDITION   CONDITION   CO //
//----------------------------------------------------------------------------//
A(;
L #_emc_gas_pi_vessel_pv;
L #_r_pres_vac;
<R;
);






    //============================= TRAN FOOTER ==============================//
    // Transition jump control:                                               //
    //------------------------------------------------------------------------//
    A     #sqSequencer.STEP.JumpCtrl;
    S     #sqSequencer.STEP.Jump;
    S     #sqSequencer.STEP.jumpDone[02];

NETWORK
TITLE =S002:t002::TRANS-v: EXIT TRANSITION AND READY THE NEXT STEP
    //------------------------------------------------------------------------//
    // Check the jump flag and jump to the next step if the transition        //
    // condition is true and has set the jump flag:                           //
    //------------------------------------------------------------------------//
    A     #sqSequencer.STEP.Jump;
    JCN   x002;

    R     #sqSequencer.STEP.Jump;
    R     #sqSequencer.STEP.Finished;

    L     04;     // Load next STEPNO to jump to if transition satisfied
    T     #sqSequencer.STEP.NumberNext; //Next Step04.

    JU    COMM;              // Transition satisfied, Exit, go to next step
x002: NOP   0;






    //============================= TRAN HEADER ==============================//
    // AUTOCODE   AUTOCODE   AUTOCODE   AUTOCODE   AUTOCODE   AUTOCODE   AUTO //
    // Bypass transition if manual jump:                                      //
    //------------------------------------------------------------------------//
    A     #sqSequencer.STEP.Finished;
    A     #smc.TRN_AND_JUMP;     //Manual jump is set Transition as bypassed
    JCN   COMM;              //exit

NETWORK
TITLE =S002::STEP 002:TRAN 003: Timer expired?
//----------------------------------------------------------------------------//
// TRAN   TRAN   TRAN   TRAN   TRAN   TRAN   TRAN   TRAN   TRAN   TRAN   TRAN //
// TRAN   TRAN   TRAN   TRAN   TRAN   TRAN   TRAN   TRAN   TRAN   TRAN   TRAN //
//----------------------------------------------------------------------------//
// Vacuum timer expired.
//----------------------------------------------------------------------------//
// CONDITION   CONDITION   CONDITION   CONDITION   CONDITION   CONDITION   CO //
// CONDITION   CONDITION   CONDITION   CONDITION   CONDITION   CONDITION   CO //
//----------------------------------------------------------------------------//
A #SQ_TIMER.Q;






    //============================= TRAN FOOTER ==============================//
    // Transition jump control:                                               //
    //------------------------------------------------------------------------//
    A     #sqSequencer.STEP.JumpCtrl;
    S     #sqSequencer.STEP.Jump;
    S     #sqSequencer.STEP.jumpDone[02];

NETWORK
TITLE =S002:t003::TRANS-v: EXIT TRANSITION AND READY THE NEXT STEP
    //------------------------------------------------------------------------//
    // Check the jump flag and jump to the next step if the transition        //
    // condition is true and has set the jump flag:                           //
    //------------------------------------------------------------------------//
    A     #sqSequencer.STEP.Jump;
    JCN   x003;

    R     #sqSequencer.STEP.Jump;
    R     #sqSequencer.STEP.Finished;

    L     03;     // Load next STEPNO to jump to if transition satisfied
    T     #sqSequencer.STEP.NumberNext; //Next Step03.

    JU    COMM;              // Transition satisfied, Exit, go to next step
x003: NOP   0;






NETWORK
TITLE =S002::STEP-002:EXIT TRANSITION:
    //========================== STEP TRANSFER ===============================//
    // Jump to the common step progression code:                              //
    //------------------------------------------------------------------------//
    JU    COMM;






NETWORK
TITLE =S003: STEP-03::UO_MX_SIP : Evacuation failed
    //================================ STEP HEADER ===========================//
    // STEP003 STEP003 STEP003 STEP003
    // AUTOCODE   AUTOCODE   AUTOCODE   AUTOCODE   AUTOCODE   AUTOCODE   AUTO //
    // STEP003 STEP003 STEP003 STEP003
    //------------------------------------------------------------------------//
    // Raise vacuum failed message.
    // Log vacuum time failed.
    // Prompt operator to confirm to try again.
    //------------------------------------------------------------------------//
S003: NOP   0;

      SET;
      R     #sqSequencer.STEP.jumpDone[03];
      A     #sqSequencer.CMD.Pause; //If paused jump
      JC    COMM;

NETWORK
TITLE =S003:STEP-03:Begin Action

      A     #sqSequencer.STEP.Finished;
      JC    A003; // Exit Action code, Jump to A003 Transition code

      //----------------------------------------------------------------------//
      // Begin step Action:                                                   //
      //----------------------------------------------------------------------//
      A     #sqSequencer.STEP.Active;
      JC    L003; // Action number loaded, Jump to L003--Step Action List

      //----------------------------------------------------------------------//
      // Load Default/Initial Step action number:                             //
      //----------------------------------------------------------------------//
      S     #sqSequencer.STEP.Active;
      S     #sqStepTimer.IN;
      L     1; //First Action, Step must contain Minimum one action
      T     #sqSequencer.STEP.ActionNumber;

//----------------------------------------------------------------------------//
// Step action list.                                                          //
// aann=mini Action step number(aa) inside main step number(nn)               //
// First Action aa00, Second action ab00, Third ac00, etc.                    //
//----------------------------------------------------------------------------//
L003: NOP   0;

      L     #sqSequencer.STEP.ActionNumber;
      JL    r003; //Wrong Action number
      JU    _003; //Action error handling
       JU    aa03; //ACTION-01


//----------------------------------------------------------------------------//
// More step action in the list can be inserted here, upto ab is tested:      //
//----------------------------------------------------------------------------//
r003: NOP   0; //Wrong action number
      S     #sqSequencer.Error_Fault;
      JU    k003; //Exit
_003: NOP   0; // Action error handling
      JU    k003; // Exit






NETWORK
TITLE =S003:: STEP-003:: : ACTION CODE
    //================================ ACT HEADER ============================//
    // ACTION ACTION ACTION ACTION ACTION ACTION ACTION ACTION ACTION ACTION  //
    // AUTOCODE   AUTOCODE   AUTOCODE   AUTOCODE   AUTOCODE   AUTOCODE   AUTO //
    // ACTION ACTION ACTION ACTION ACTION ACTION ACTION ACTION ACTION ACTION  //
    //------------------------------------------------------------------------//
    // //Raise vacuum failed message.
    // //Log vacuum time failed.
    // //Prompt operator to confirm to try again.
    aa03: NOP   0;

    //------------------------------------------------------------------------//
    // ACT ACT ACT ACT ACT ACT ACT ACT ACT ACT ACT ACT ACT ACT ACT ACT ACT    //
    //------------------------------------------------------------------------//
    //Log time vacuum failed
SET;
S #_log_msg_vacuum_fail;
S #_prompt_try_again;

    //------------------------------------------------------------------------//
    // VERIFY  VERIFY VERIFY VERIFY VERIFY VERIFY VERIFY VERIFY VERIFY VERIFY //
    //------------------------------------------------------------------------//
    A "uncondJump";
    S     #sqSequencer.STEP.ActionVerified; //Action verified

    //------------------------------------------------------------------------//
    // Action done:                                                           //
    //------------------------------------------------------------------------//
    O     #sqSequencer.STEP.ActionVerified;
    O     #smc.NO_VERIFIC;       //No verification , bypass verification code
    S     #sqSequencer.STEP.ActionFinished;






    //============================= STEP FOOTER ==============================//
    // AUTOCODE   AUTOCODE   AUTOCODE   AUTOCODE   AUTOCODE   AUTOCODE   AUTO //
    // Get Ready after action finished:                                       //
    //------------------------------------------------------------------------//
    A     #sqSequencer.STEP.ActionFinished;
    JCN   k003;

    //------------------------------------------------------------------------//
    // Reset Action finished flag, ready for next step action:                //
    //------------------------------------------------------------------------//
    R     #sqSequencer.STEP.ActionVerified;
    R     #sqSequencer.STEP.ActionFinished;

    //------------------------------------------------------------------------//
    // If ALL actions are finished:                                           //
    //------------------------------------------------------------------------//
    SET   ;
    S     #sqSequencer.STEP.Finished;
    R     #sqSequencer.STEP.Active;
    S     #sqSequencer.STEP.Done[03];

    //------------------------------------------------------------------------//
    // End Step action(s):                                                    //
    //------------------------------------------------------------------------//
    JU    k003;

//----------------------------------------------------------------------------//
// Finished Step Action(s):                                                   //
//----------------------------------------------------------------------------//
k003: NOP   0;

    A     #sqStepTimerExpired;
    S     #sqSequencer.STEP.WithError[03]; // Step error flag
    S     #sqSequencer.Error_Fault;
    R     #sqStepTimer.IN;

NETWORK
TITLE =S003:STEP-003::Begin Transition
    //------------------------------------------------------------------------//
    // Begin the transition code:                                             //
    //------------------------------------------------------------------------//
    A003: NOP   0;
    R     #sqStepTimer.IN;






    //============================= TRAN HEADER ==============================//
    // AUTOCODE   AUTOCODE   AUTOCODE   AUTOCODE   AUTOCODE   AUTOCODE   AUTO //
    // Bypass transition if manual jump:                                      //
    //------------------------------------------------------------------------//
    A     #sqSequencer.STEP.Finished;
    A     #smc.TRN_AND_JUMP;     //Manual jump is set Transition as bypassed
    JCN   COMM;              //exit

NETWORK
TITLE =S003::STEP 003:TRAN 004: Try again?
//----------------------------------------------------------------------------//
// TRAN   TRAN   TRAN   TRAN   TRAN   TRAN   TRAN   TRAN   TRAN   TRAN   TRAN //
// TRAN   TRAN   TRAN   TRAN   TRAN   TRAN   TRAN   TRAN   TRAN   TRAN   TRAN //
//----------------------------------------------------------------------------//
// Operator want to try again.
//----------------------------------------------------------------------------//
// CONDITION   CONDITION   CONDITION   CONDITION   CONDITION   CONDITION   CO //
// CONDITION   CONDITION   CONDITION   CONDITION   CONDITION   CONDITION   CO //
//----------------------------------------------------------------------------//
A #_prompt_try_again_confirm_yes;






    //============================= TRAN FOOTER ==============================//
    // Transition jump control:                                               //
    //------------------------------------------------------------------------//
    A     #sqSequencer.STEP.JumpCtrl;
    S     #sqSequencer.STEP.Jump;
    S     #sqSequencer.STEP.jumpDone[03];

NETWORK
TITLE =S003:t004::TRANS-v: EXIT TRANSITION AND READY THE NEXT STEP
    //------------------------------------------------------------------------//
    // Check the jump flag and jump to the next step if the transition        //
    // condition is true and has set the jump flag:                           //
    //------------------------------------------------------------------------//
    A     #sqSequencer.STEP.Jump;
    JCN   x004;

    R     #sqSequencer.STEP.Jump;
    R     #sqSequencer.STEP.Finished;

    L     05;     // Load next STEPNO to jump to if transition satisfied
    T     #sqSequencer.STEP.NumberNext; //Next Step05.

    JU    COMM;              // Transition satisfied, Exit, go to next step
x004: NOP   0;






    //============================= TRAN HEADER ==============================//
    // AUTOCODE   AUTOCODE   AUTOCODE   AUTOCODE   AUTOCODE   AUTOCODE   AUTO //
    // Bypass transition if manual jump:                                      //
    //------------------------------------------------------------------------//
    A     #sqSequencer.STEP.Finished;
    A     #smc.TRN_AND_JUMP;     //Manual jump is set Transition as bypassed
    JCN   COMM;              //exit

NETWORK
TITLE =S003::STEP 003:TRAN 005: No try?
//----------------------------------------------------------------------------//
// TRAN   TRAN   TRAN   TRAN   TRAN   TRAN   TRAN   TRAN   TRAN   TRAN   TRAN //
// TRAN   TRAN   TRAN   TRAN   TRAN   TRAN   TRAN   TRAN   TRAN   TRAN   TRAN //
//----------------------------------------------------------------------------//
// Operator don't want to try again.
//----------------------------------------------------------------------------//
// CONDITION   CONDITION   CONDITION   CONDITION   CONDITION   CONDITION   CO //
// CONDITION   CONDITION   CONDITION   CONDITION   CONDITION   CONDITION   CO //
//----------------------------------------------------------------------------//
A #_prompt_try_again_confirm_no;






    //============================= TRAN FOOTER ==============================//
    // Transition jump control:                                               //
    //------------------------------------------------------------------------//
    A     #sqSequencer.STEP.JumpCtrl;
    S     #sqSequencer.STEP.Jump;
    S     #sqSequencer.STEP.jumpDone[03];

NETWORK
TITLE =S003:t005::TRANS-v: EXIT TRANSITION AND READY THE NEXT STEP
    //------------------------------------------------------------------------//
    // Check the jump flag and jump to the next step if the transition        //
    // condition is true and has set the jump flag:                           //
    //------------------------------------------------------------------------//
    A     #sqSequencer.STEP.Jump;
    JCN   x005;

    R     #sqSequencer.STEP.Jump;
    R     #sqSequencer.STEP.Finished;

    L     06;     // Load next STEPNO to jump to if transition satisfied
    T     #sqSequencer.STEP.NumberNext; //Next Step06.

    JU    COMM;              // Transition satisfied, Exit, go to next step
x005: NOP   0;






NETWORK
TITLE =S003::STEP-003:EXIT TRANSITION:
    //========================== STEP TRANSFER ===============================//
    // Jump to the common step progression code:                              //
    //------------------------------------------------------------------------//
    JU    COMM;






NETWORK
TITLE =S004: STEP-04::UO_MX_SIP : Vacuum operation finished.
    //================================ STEP HEADER ===========================//
    // STEP004 STEP004 STEP004 STEP004
    // AUTOCODE   AUTOCODE   AUTOCODE   AUTOCODE   AUTOCODE   AUTOCODE   AUTO //
    // STEP004 STEP004 STEP004 STEP004
    //------------------------------------------------------------------------//
    // Close Mx vacuum valves.
    //------------------------------------------------------------------------//
S004: NOP   0;

      SET;
      R     #sqSequencer.STEP.jumpDone[04];
      A     #sqSequencer.CMD.Pause; //If paused jump
      JC    COMM;

NETWORK
TITLE =S004:STEP-04:Begin Action

      A     #sqSequencer.STEP.Finished;
      JC    A004; // Exit Action code, Jump to A004 Transition code

      //----------------------------------------------------------------------//
      // Begin step Action:                                                   //
      //----------------------------------------------------------------------//
      A     #sqSequencer.STEP.Active;
      JC    L004; // Action number loaded, Jump to L004--Step Action List

      //----------------------------------------------------------------------//
      // Load Default/Initial Step action number:                             //
      //----------------------------------------------------------------------//
      S     #sqSequencer.STEP.Active;
      S     #sqStepTimer.IN;
      L     1; //First Action, Step must contain Minimum one action
      T     #sqSequencer.STEP.ActionNumber;

//----------------------------------------------------------------------------//
// Step action list.                                                          //
// aann=mini Action step number(aa) inside main step number(nn)               //
// First Action aa00, Second action ab00, Third ac00, etc.                    //
//----------------------------------------------------------------------------//
L004: NOP   0;

      L     #sqSequencer.STEP.ActionNumber;
      JL    r004; //Wrong Action number
      JU    _004; //Action error handling
       JU    aa04; //ACTION-01
JU    ab04; //ACTION-02


//----------------------------------------------------------------------------//
// More step action in the list can be inserted here, upto ab is tested:      //
//----------------------------------------------------------------------------//
r004: NOP   0; //Wrong action number
      S     #sqSequencer.Error_Fault;
      JU    k004; //Exit
_004: NOP   0; // Action error handling
      JU    k004; // Exit






NETWORK
TITLE =S004:: STEP-004:: : ACTION CODE
    //================================ ACT HEADER ============================//
    // ACTION ACTION ACTION ACTION ACTION ACTION ACTION ACTION ACTION ACTION  //
    // AUTOCODE   AUTOCODE   AUTOCODE   AUTOCODE   AUTOCODE   AUTOCODE   AUTO //
    // ACTION ACTION ACTION ACTION ACTION ACTION ACTION ACTION ACTION ACTION  //
    //------------------------------------------------------------------------//
    // //Close Mx Vacuum Valve.
    aa04: NOP   0;

    //------------------------------------------------------------------------//
    // ACT ACT ACT ACT ACT ACT ACT ACT ACT ACT ACT ACT ACT ACT ACT ACT ACT    //
    //------------------------------------------------------------------------//
    //Close vacuum valve.
L "dbCONST".SEL.GAS.NONE;
T #_emc_gas_medium_gas;
L "dbCONST".BLK.CMD.RESTART;
T #_emc_gas_cmd;

// Stop timer
SET;
R #sqSeqTimerStart;

    //------------------------------------------------------------------------//
    // VERIFY  VERIFY VERIFY VERIFY VERIFY VERIFY VERIFY VERIFY VERIFY VERIFY //
    //------------------------------------------------------------------------//
    A(;
L   #_emc_gas_state;
L   "dbCONST".BLK.STATE.STOPPED;
>I;
);
A(;
L   #_emc_gas_state;
L   "dbCONST".BLK.STATE.INTERLOCKED;
<I;
);
    S     #sqSequencer.STEP.ActionVerified; //Action verified

    //------------------------------------------------------------------------//
    // Action done:                                                           //
    //------------------------------------------------------------------------//
    O     #sqSequencer.STEP.ActionVerified;
    O     #smc.NO_VERIFIC;       //No verification , bypass verification code
    S     #sqSequencer.STEP.ActionFinished;






    //============================= ACT FOOTER ===============================//
    // AUTOCODE   AUTOCODE   AUTOCODE   AUTOCODE   AUTOCODE   AUTOCODE   AUTO //
    // Get Ready after action finished:                                       //
    //------------------------------------------------------------------------//
    A     #sqSequencer.STEP.ActionFinished;
    JCN   k004;

    //------------------------------------------------------------------------//
    // Reset Action finished flag, ready for next step action:                //
    //------------------------------------------------------------------------//
    R     #sqSequencer.STEP.ActionVerified;
    R     #sqSequencer.STEP.ActionFinished;

    //------------------------------------------------------------------------//
    // Load Next Step Action number:                                          //
    //------------------------------------------------------------------------//
    L     02; //Load next Action
    T     #sqSequencer.STEP.ActionNumber;






NETWORK
TITLE =S004:: STEP-004:: : ACTION CODE
    //================================ ACT HEADER ============================//
    // ACTION ACTION ACTION ACTION ACTION ACTION ACTION ACTION ACTION ACTION  //
    // AUTOCODE   AUTOCODE   AUTOCODE   AUTOCODE   AUTOCODE   AUTOCODE   AUTO //
    // ACTION ACTION ACTION ACTION ACTION ACTION ACTION ACTION ACTION ACTION  //
    //------------------------------------------------------------------------//
    // //Clear the EMC restart command
    ab04: NOP   0;

    //------------------------------------------------------------------------//
    // ACT ACT ACT ACT ACT ACT ACT ACT ACT ACT ACT ACT ACT ACT ACT ACT ACT    //
    //------------------------------------------------------------------------//
    L "dbCONST".BLK.CMD.START;
T #_emc_gas_cmd;

    //------------------------------------------------------------------------//
    // VERIFY  VERIFY VERIFY VERIFY VERIFY VERIFY VERIFY VERIFY VERIFY VERIFY //
    //------------------------------------------------------------------------//

    S     #sqSequencer.STEP.ActionVerified; //Action verified

    //------------------------------------------------------------------------//
    // Action done:                                                           //
    //------------------------------------------------------------------------//
    O     #sqSequencer.STEP.ActionVerified;
    O     #smc.NO_VERIFIC;       //No verification , bypass verification code
    S     #sqSequencer.STEP.ActionFinished;






    //============================= STEP FOOTER ==============================//
    // AUTOCODE   AUTOCODE   AUTOCODE   AUTOCODE   AUTOCODE   AUTOCODE   AUTO //
    // Get Ready after action finished:                                       //
    //------------------------------------------------------------------------//
    A     #sqSequencer.STEP.ActionFinished;
    JCN   k004;

    //------------------------------------------------------------------------//
    // Reset Action finished flag, ready for next step action:                //
    //------------------------------------------------------------------------//
    R     #sqSequencer.STEP.ActionVerified;
    R     #sqSequencer.STEP.ActionFinished;

    //------------------------------------------------------------------------//
    // If ALL actions are finished:                                           //
    //------------------------------------------------------------------------//
    SET   ;
    S     #sqSequencer.STEP.Finished;
    R     #sqSequencer.STEP.Active;
    S     #sqSequencer.STEP.Done[04];

    //------------------------------------------------------------------------//
    // End Step action(s):                                                    //
    //------------------------------------------------------------------------//
    JU    k004;

//----------------------------------------------------------------------------//
// Finished Step Action(s):                                                   //
//----------------------------------------------------------------------------//
k004: NOP   0;

    A     #sqStepTimerExpired;
    S     #sqSequencer.STEP.WithError[04]; // Step error flag
    S     #sqSequencer.Error_Fault;
    R     #sqStepTimer.IN;

NETWORK
TITLE =S004:STEP-004::Begin Transition
    //------------------------------------------------------------------------//
    // Begin the transition code:                                             //
    //------------------------------------------------------------------------//
    A004: NOP   0;
    R     #sqStepTimer.IN;






    //============================= TRAN HEADER ==============================//
    // AUTOCODE   AUTOCODE   AUTOCODE   AUTOCODE   AUTOCODE   AUTOCODE   AUTO //
    // Bypass transition if manual jump:                                      //
    //------------------------------------------------------------------------//
    A     #sqSequencer.STEP.Finished;
    A     #smc.TRN_AND_JUMP;     //Manual jump is set Transition as bypassed
    JCN   COMM;              //exit

NETWORK
TITLE =S004::STEP 004:TRAN 006: All Vacuum operations complete
//----------------------------------------------------------------------------//
// TRAN   TRAN   TRAN   TRAN   TRAN   TRAN   TRAN   TRAN   TRAN   TRAN   TRAN //
// TRAN   TRAN   TRAN   TRAN   TRAN   TRAN   TRAN   TRAN   TRAN   TRAN   TRAN //
//----------------------------------------------------------------------------//
// Vacuum valve closed.
//----------------------------------------------------------------------------//
// CONDITION   CONDITION   CONDITION   CONDITION   CONDITION   CONDITION   CO //
// CONDITION   CONDITION   CONDITION   CONDITION   CONDITION   CONDITION   CO //
//----------------------------------------------------------------------------//
A(;
L 	#_emc_gas_state;
L 	"dbCONST".BLK.STATE.COMPLETED;
==I;
);






    //============================= TRAN FOOTER ==============================//
    // Transition jump control:                                               //
    //------------------------------------------------------------------------//
    A     #sqSequencer.STEP.JumpCtrl;
    S     #sqSequencer.STEP.Jump;
    S     #sqSequencer.STEP.jumpDone[04];

NETWORK
TITLE =S004:t006::TRANS-v: EXIT TRANSITION AND READY THE NEXT STEP
    //------------------------------------------------------------------------//
    // Check the jump flag and jump to the next step if the transition        //
    // condition is true and has set the jump flag:                           //
    //------------------------------------------------------------------------//
    A     #sqSequencer.STEP.Jump;
    JCN   x006;

    R     #sqSequencer.STEP.Jump;
    R     #sqSequencer.STEP.Finished;

    L     07;     // Load next STEPNO to jump to if transition satisfied
    T     #sqSequencer.STEP.NumberNext; //Next Step07.

    JU    COMM;              // Transition satisfied, Exit, go to next step
x006: NOP   0;






NETWORK
TITLE =S004::STEP-004:EXIT TRANSITION:
    //========================== STEP TRANSFER ===============================//
    // Jump to the common step progression code:                              //
    //------------------------------------------------------------------------//
    JU    COMM;






NETWORK
TITLE =S005: STEP-05::UO_MX_SIP : Log Operator Repeat
    //================================ STEP HEADER ===========================//
    // STEP005 STEP005 STEP005 STEP005
    // AUTOCODE   AUTOCODE   AUTOCODE   AUTOCODE   AUTOCODE   AUTOCODE   AUTO //
    // STEP005 STEP005 STEP005 STEP005
    //------------------------------------------------------------------------//
    // Log operator repeat.
    //------------------------------------------------------------------------//
S005: NOP   0;

      SET;
      R     #sqSequencer.STEP.jumpDone[05];
      A     #sqSequencer.CMD.Pause; //If paused jump
      JC    COMM;

NETWORK
TITLE =S005:STEP-05:Begin Action

      A     #sqSequencer.STEP.Finished;
      JC    A005; // Exit Action code, Jump to A005 Transition code

      //----------------------------------------------------------------------//
      // Begin step Action:                                                   //
      //----------------------------------------------------------------------//
      A     #sqSequencer.STEP.Active;
      JC    L005; // Action number loaded, Jump to L005--Step Action List

      //----------------------------------------------------------------------//
      // Load Default/Initial Step action number:                             //
      //----------------------------------------------------------------------//
      S     #sqSequencer.STEP.Active;
      S     #sqStepTimer.IN;
      L     1; //First Action, Step must contain Minimum one action
      T     #sqSequencer.STEP.ActionNumber;

//----------------------------------------------------------------------------//
// Step action list.                                                          //
// aann=mini Action step number(aa) inside main step number(nn)               //
// First Action aa00, Second action ab00, Third ac00, etc.                    //
//----------------------------------------------------------------------------//
L005: NOP   0;

      L     #sqSequencer.STEP.ActionNumber;
      JL    r005; //Wrong Action number
      JU    _005; //Action error handling
       JU    aa05; //ACTION-01


//----------------------------------------------------------------------------//
// More step action in the list can be inserted here, upto ab is tested:      //
//----------------------------------------------------------------------------//
r005: NOP   0; //Wrong action number
      S     #sqSequencer.Error_Fault;
      JU    k005; //Exit
_005: NOP   0; // Action error handling
      JU    k005; // Exit






NETWORK
TITLE =S005:: STEP-005:: : ACTION CODE
    //================================ ACT HEADER ============================//
    // ACTION ACTION ACTION ACTION ACTION ACTION ACTION ACTION ACTION ACTION  //
    // AUTOCODE   AUTOCODE   AUTOCODE   AUTOCODE   AUTOCODE   AUTOCODE   AUTO //
    // ACTION ACTION ACTION ACTION ACTION ACTION ACTION ACTION ACTION ACTION  //
    //------------------------------------------------------------------------//
    // //Log operator repeat.
    aa05: NOP   0;

    //------------------------------------------------------------------------//
    // ACT ACT ACT ACT ACT ACT ACT ACT ACT ACT ACT ACT ACT ACT ACT ACT ACT    //
    //------------------------------------------------------------------------//
    //Log operator repeat.
SET;
S #_log_msg_vacuum_fail_repeat;
R #_prompt_try_again_confirm_yes;

    //------------------------------------------------------------------------//
    // VERIFY  VERIFY VERIFY VERIFY VERIFY VERIFY VERIFY VERIFY VERIFY VERIFY //
    //------------------------------------------------------------------------//
    A "uncondJump";
    S     #sqSequencer.STEP.ActionVerified; //Action verified

    //------------------------------------------------------------------------//
    // Action done:                                                           //
    //------------------------------------------------------------------------//
    O     #sqSequencer.STEP.ActionVerified;
    O     #smc.NO_VERIFIC;       //No verification , bypass verification code
    S     #sqSequencer.STEP.ActionFinished;






    //============================= STEP FOOTER ==============================//
    // AUTOCODE   AUTOCODE   AUTOCODE   AUTOCODE   AUTOCODE   AUTOCODE   AUTO //
    // Get Ready after action finished:                                       //
    //------------------------------------------------------------------------//
    A     #sqSequencer.STEP.ActionFinished;
    JCN   k005;

    //------------------------------------------------------------------------//
    // Reset Action finished flag, ready for next step action:                //
    //------------------------------------------------------------------------//
    R     #sqSequencer.STEP.ActionVerified;
    R     #sqSequencer.STEP.ActionFinished;

    //------------------------------------------------------------------------//
    // If ALL actions are finished:                                           //
    //------------------------------------------------------------------------//
    SET   ;
    S     #sqSequencer.STEP.Finished;
    R     #sqSequencer.STEP.Active;
    S     #sqSequencer.STEP.Done[05];

    //------------------------------------------------------------------------//
    // End Step action(s):                                                    //
    //------------------------------------------------------------------------//
    JU    k005;

//----------------------------------------------------------------------------//
// Finished Step Action(s):                                                   //
//----------------------------------------------------------------------------//
k005: NOP   0;

    A     #sqStepTimerExpired;
    S     #sqSequencer.STEP.WithError[05]; // Step error flag
    S     #sqSequencer.Error_Fault;
    R     #sqStepTimer.IN;

NETWORK
TITLE =S005:STEP-005::Begin Transition
    //------------------------------------------------------------------------//
    // Begin the transition code:                                             //
    //------------------------------------------------------------------------//
    A005: NOP   0;
    R     #sqStepTimer.IN;






    //============================= TRAN HEADER ==============================//
    // AUTOCODE   AUTOCODE   AUTOCODE   AUTOCODE   AUTOCODE   AUTOCODE   AUTO //
    // Bypass transition if manual jump:                                      //
    //------------------------------------------------------------------------//
    A     #sqSequencer.STEP.Finished;
    A     #smc.TRN_AND_JUMP;     //Manual jump is set Transition as bypassed
    JCN   COMM;              //exit

NETWORK
TITLE =S005::STEP 005:TRAN 007: Empty Transition
//----------------------------------------------------------------------------//
// TRAN   TRAN   TRAN   TRAN   TRAN   TRAN   TRAN   TRAN   TRAN   TRAN   TRAN //
// TRAN   TRAN   TRAN   TRAN   TRAN   TRAN   TRAN   TRAN   TRAN   TRAN   TRAN //
//----------------------------------------------------------------------------//
// Empty Transition
//----------------------------------------------------------------------------//
// CONDITION   CONDITION   CONDITION   CONDITION   CONDITION   CONDITION   CO //
// CONDITION   CONDITION   CONDITION   CONDITION   CONDITION   CONDITION   CO //
//----------------------------------------------------------------------------//
A "uncondJump";






    //============================= TRAN FOOTER ==============================//
    // Transition jump control:                                               //
    //------------------------------------------------------------------------//
    A     #sqSequencer.STEP.JumpCtrl;
    S     #sqSequencer.STEP.Jump;
    S     #sqSequencer.STEP.jumpDone[05];

NETWORK
TITLE =S005:t007::TRANS-v: EXIT TRANSITION AND READY THE NEXT STEP
    //------------------------------------------------------------------------//
    // Check the jump flag and jump to the next step if the transition        //
    // condition is true and has set the jump flag:                           //
    //------------------------------------------------------------------------//
    A     #sqSequencer.STEP.Jump;
    JCN   x007;

    R     #sqSequencer.STEP.Jump;
    R     #sqSequencer.STEP.Finished;

    L     02;     // Load next STEPNO to jump to if transition satisfied
    T     #sqSequencer.STEP.NumberNext; //Next Step02.

    JU    COMM;              // Transition satisfied, Exit, go to next step
x007: NOP   0;






NETWORK
TITLE =S005::STEP-005:EXIT TRANSITION:
    //========================== STEP TRANSFER ===============================//
    // Jump to the common step progression code:                              //
    //------------------------------------------------------------------------//
    JU    COMM;






NETWORK
TITLE =S006: STEP-06::UO_MX_SIP : Log Operator Abort
    //================================ STEP HEADER ===========================//
    // STEP006 STEP006 STEP006 STEP006
    // AUTOCODE   AUTOCODE   AUTOCODE   AUTOCODE   AUTOCODE   AUTOCODE   AUTO //
    // STEP006 STEP006 STEP006 STEP006
    //------------------------------------------------------------------------//
    // Set devices to safe state.
    // Log operator abort.
    //------------------------------------------------------------------------//
S006: NOP   0;

      SET;
      R     #sqSequencer.STEP.jumpDone[06];
      A     #sqSequencer.CMD.Pause; //If paused jump
      JC    COMM;

NETWORK
TITLE =S006:STEP-06:Begin Action

      A     #sqSequencer.STEP.Finished;
      JC    A006; // Exit Action code, Jump to A006 Transition code

      //----------------------------------------------------------------------//
      // Begin step Action:                                                   //
      //----------------------------------------------------------------------//
      A     #sqSequencer.STEP.Active;
      JC    L006; // Action number loaded, Jump to L006--Step Action List

      //----------------------------------------------------------------------//
      // Load Default/Initial Step action number:                             //
      //----------------------------------------------------------------------//
      S     #sqSequencer.STEP.Active;
      S     #sqStepTimer.IN;
      L     1; //First Action, Step must contain Minimum one action
      T     #sqSequencer.STEP.ActionNumber;

//----------------------------------------------------------------------------//
// Step action list.                                                          //
// aann=mini Action step number(aa) inside main step number(nn)               //
// First Action aa00, Second action ab00, Third ac00, etc.                    //
//----------------------------------------------------------------------------//
L006: NOP   0;

      L     #sqSequencer.STEP.ActionNumber;
      JL    r006; //Wrong Action number
      JU    _006; //Action error handling
       JU    aa06; //ACTION-01


//----------------------------------------------------------------------------//
// More step action in the list can be inserted here, upto ab is tested:      //
//----------------------------------------------------------------------------//
r006: NOP   0; //Wrong action number
      S     #sqSequencer.Error_Fault;
      JU    k006; //Exit
_006: NOP   0; // Action error handling
      JU    k006; // Exit






NETWORK
TITLE =S006:: STEP-006:: : ACTION CODE
    //================================ ACT HEADER ============================//
    // ACTION ACTION ACTION ACTION ACTION ACTION ACTION ACTION ACTION ACTION  //
    // AUTOCODE   AUTOCODE   AUTOCODE   AUTOCODE   AUTOCODE   AUTOCODE   AUTO //
    // ACTION ACTION ACTION ACTION ACTION ACTION ACTION ACTION ACTION ACTION  //
    //------------------------------------------------------------------------//
    // //Log operator abort.
    aa06: NOP   0;

    //------------------------------------------------------------------------//
    // ACT ACT ACT ACT ACT ACT ACT ACT ACT ACT ACT ACT ACT ACT ACT ACT ACT    //
    //------------------------------------------------------------------------//
    //Log operator abort.
SET;
S #_log_msg_vacuum_fail_abort;
R #_prompt_try_again_confirm_no;
S #smc.ABORTED;

// Set all used equipment to safe state.
L "dbCONST".BLK.CMD.STOP;
T #_emv_vessel_cmd;
T #_emv_inlet_cmd;
T #_emg_filter_cmd;
T  #_emc_gas_cmd;
T  #_emc_water_cmd;
T  #_emx_drain_cmd;
T  #_emx_mmfl_cmd;

    //------------------------------------------------------------------------//
    // VERIFY  VERIFY VERIFY VERIFY VERIFY VERIFY VERIFY VERIFY VERIFY VERIFY //
    //------------------------------------------------------------------------//
    A "uncondJump";
    S     #sqSequencer.STEP.ActionVerified; //Action verified

    //------------------------------------------------------------------------//
    // Action done:                                                           //
    //------------------------------------------------------------------------//
    O     #sqSequencer.STEP.ActionVerified;
    O     #smc.NO_VERIFIC;       //No verification , bypass verification code
    S     #sqSequencer.STEP.ActionFinished;






    //============================= STEP FOOTER ==============================//
    // AUTOCODE   AUTOCODE   AUTOCODE   AUTOCODE   AUTOCODE   AUTOCODE   AUTO //
    // Get Ready after action finished:                                       //
    //------------------------------------------------------------------------//
    A     #sqSequencer.STEP.ActionFinished;
    JCN   k006;

    //------------------------------------------------------------------------//
    // Reset Action finished flag, ready for next step action:                //
    //------------------------------------------------------------------------//
    R     #sqSequencer.STEP.ActionVerified;
    R     #sqSequencer.STEP.ActionFinished;

    //------------------------------------------------------------------------//
    // If ALL actions are finished:                                           //
    //------------------------------------------------------------------------//
    SET   ;
    S     #sqSequencer.STEP.Finished;
    R     #sqSequencer.STEP.Active;
    S     #sqSequencer.STEP.Done[06];

    //------------------------------------------------------------------------//
    // End Step action(s):                                                    //
    //------------------------------------------------------------------------//
    JU    k006;

//----------------------------------------------------------------------------//
// Finished Step Action(s):                                                   //
//----------------------------------------------------------------------------//
k006: NOP   0;

    A     #sqStepTimerExpired;
    S     #sqSequencer.STEP.WithError[06]; // Step error flag
    S     #sqSequencer.Error_Fault;
    R     #sqStepTimer.IN;

NETWORK
TITLE =S006:STEP-006::Begin Transition
    //------------------------------------------------------------------------//
    // Begin the transition code:                                             //
    //------------------------------------------------------------------------//
    A006: NOP   0;
    R     #sqStepTimer.IN;






    //============================= TRAN HEADER ==============================//
    // AUTOCODE   AUTOCODE   AUTOCODE   AUTOCODE   AUTOCODE   AUTOCODE   AUTO //
    // Bypass transition if manual jump:                                      //
    //------------------------------------------------------------------------//
    A     #sqSequencer.STEP.Finished;
    A     #smc.TRN_AND_JUMP;     //Manual jump is set Transition as bypassed
    JCN   COMM;              //exit

NETWORK
TITLE =S006::STEP 006:TRAN 008: Empty Transition
//----------------------------------------------------------------------------//
// TRAN   TRAN   TRAN   TRAN   TRAN   TRAN   TRAN   TRAN   TRAN   TRAN   TRAN //
// TRAN   TRAN   TRAN   TRAN   TRAN   TRAN   TRAN   TRAN   TRAN   TRAN   TRAN //
//----------------------------------------------------------------------------//
// Empty Transition
//----------------------------------------------------------------------------//
// CONDITION   CONDITION   CONDITION   CONDITION   CONDITION   CONDITION   CO //
// CONDITION   CONDITION   CONDITION   CONDITION   CONDITION   CONDITION   CO //
//----------------------------------------------------------------------------//
A "uncondJump";






    //============================= TRAN FOOTER ==============================//
    // Transition jump control:                                               //
    //------------------------------------------------------------------------//
    A     #sqSequencer.STEP.JumpCtrl;
    S     #sqSequencer.STEP.Jump;
    S     #sqSequencer.STEP.jumpDone[06];

NETWORK
TITLE =S006:t008::TRANS-v: EXIT TRANSITION AND READY THE NEXT STEP
    //------------------------------------------------------------------------//
    // Check the jump flag and jump to the next step if the transition        //
    // condition is true and has set the jump flag:                           //
    //------------------------------------------------------------------------//
    A     #sqSequencer.STEP.Jump;
    JCN   x008;

    R     #sqSequencer.STEP.Jump;
    R     #sqSequencer.STEP.Finished;

    L     25;     // Load next STEPNO to jump to if transition satisfied
    T     #sqSequencer.STEP.NumberNext; //Next Step25.

    JU    COMM;              // Transition satisfied, Exit, go to next step
x008: NOP   0;






NETWORK
TITLE =S006::STEP-006:EXIT TRANSITION:
    //========================== STEP TRANSFER ===============================//
    // Jump to the common step progression code:                              //
    //------------------------------------------------------------------------//
    JU    COMM;






NETWORK
TITLE =S007: STEP-07::UO_MX_SIP : Initiate MX and MMFLx SIP Operations
    //================================ STEP HEADER ===========================//
    // STEP007 STEP007 STEP007 STEP007
    // AUTOCODE   AUTOCODE   AUTOCODE   AUTOCODE   AUTOCODE   AUTOCODE   AUTO //
    // STEP007 STEP007 STEP007 STEP007
    //------------------------------------------------------------------------//
    // Open Mx steam supply on WFI/PS lines.
    //
    // Log steam opened time.
    //------------------------------------------------------------------------//
S007: NOP   0;

      SET;
      R     #sqSequencer.STEP.jumpDone[07];
      A     #sqSequencer.CMD.Pause; //If paused jump
      JC    COMM;

NETWORK
TITLE =S007:STEP-07:Begin Action

      A     #sqSequencer.STEP.Finished;
      JC    A007; // Exit Action code, Jump to A007 Transition code

      //----------------------------------------------------------------------//
      // Begin step Action:                                                   //
      //----------------------------------------------------------------------//
      A     #sqSequencer.STEP.Active;
      JC    L007; // Action number loaded, Jump to L007--Step Action List

      //----------------------------------------------------------------------//
      // Load Default/Initial Step action number:                             //
      //----------------------------------------------------------------------//
      S     #sqSequencer.STEP.Active;
      S     #sqStepTimer.IN;
      L     1; //First Action, Step must contain Minimum one action
      T     #sqSequencer.STEP.ActionNumber;

//----------------------------------------------------------------------------//
// Step action list.                                                          //
// aann=mini Action step number(aa) inside main step number(nn)               //
// First Action aa00, Second action ab00, Third ac00, etc.                    //
//----------------------------------------------------------------------------//
L007: NOP   0;

      L     #sqSequencer.STEP.ActionNumber;
      JL    r007; //Wrong Action number
      JU    _007; //Action error handling
       JU    aa07; //ACTION-01


